SUBAPPLICATION Ventilsteuerung_Uebung_020h (* DigitalInput_I1 auf DigitalOutput_Q1; E_PULSE; Impulsformend *)
  (* Standard: 61499-2 *)
  (* Version 1.0, 2023-10-23, franz *)
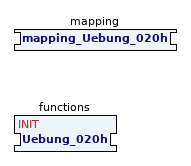
  SUBAPPS
    mapping : mapping_Uebung_020h;
    functions : Uebung_020h;
  END_SUBAPPS
END_SUBAPPLICATION
